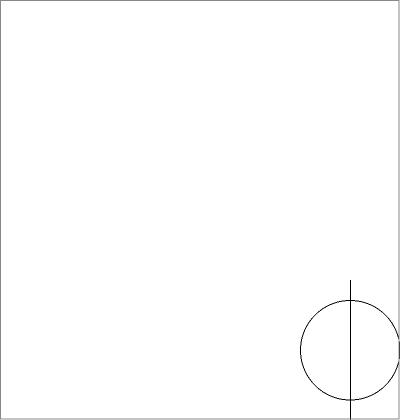
VISUALIZATION Visualization  // 400x420
    Ellipse (300,300 100x100)
        p1097714728: MAIN.rRadius * 20
    Line (350,350) (350,350)
        p3528305787: MAIN.ip1x
        p2773130477: MAIN.ip1y
        p874137650: MAIN.ip2x
        p1126004900: MAIN.ip2y
    Line (350,300) (350,420)
        p3528305787: MAIN.rStickLength + MAIN.rRadius
        p874137650: MAIN.rStickLength + MAIN.rRadius
    Line (350,280) (350,400)
        p3528305787: MAIN.rStickLength - MAIN.rRadius
        p874137650: MAIN.rStickLength - MAIN.rRadius
END_VISUALIZATION

(* stored: Version 1.1.0.1
   Visu Visualization: Id {1a5a8797-3bee-4cde-a5ac-f966e0a6c27b} *)
